Fanuc KAREL source: kt00480.KL

-- PROVISIONAL review KL for V1013-1; original PC SHA256 f996ed086115790f3e2e3a040581a68f332a77b733f2f6de9ec9aacdc0f7d8bd
-- Incomplete behavior may be omitted. Consult companion uncertainty JSON. Do not deploy.
PROGRAM KT00480
%NOLOCKGROUP
-- UNRESOLVED_DECL P1 type=000101
-- UNRESOLVED_DECL P2 type=000102
-- UNRESOLVED_DECL OUT type=000102
BEGIN
  -- UNRESOLVED_PC offsets 5-20; opcodes 2E,22,32,35
  -- UNRESOLVED_PC offsets 25-59; opcodes 49,49,7E,60,7E,4A
  -- UNRESOLVED_PC offsets 64-68; opcodes 7F
END KT00480
